INTERFACE PUBLIC LogEventFormatter EXTENDS __SYSTEM.IQueryInterface

METHOD Format : T_MaxString
VAR_INPUT
	event : LogEvent;
END_VAR
END_METHOD

END_INTERFACE

(* stored: Version 1.1.0.1
   Itf LogEventFormatter: Id {ee5ac149-1672-473c-9849-4b71bf68d930}
   Method Format: Id {36298a3b-e769-43d0-b78f-48067b72a299} *)
